// TIA Portal V20 export
TYPE "LKinCtrl_typeSetFlagElement_Bool"
   STRUCT
      flag : Int := -1;   // flag to be set
      flagMode : USInt := 1;   // (see LKinCtrl_PLC_Tags) 0: deactivated; 1: SET_BEFORE_AND_NO_RESET; 2: SET_BEFORE_AND_RESET_AFTER; 3: SET_BEFORE_AND_RESET_AFTER_ONE_CYCLE; 5: SET_BEFORE_AND_NO_RESET_AND_WAIT_FOR_ACKNOWLEDGE; 10: LKINCTRL_FM_SET_AT_REMAINING_DISTANCE; 11: LKINCTRL_FM_SET_AFTER_AND_NO_RESET; 13: LKINCTRL_FM_SET_AFTER_AND_RESET_AFTER_ONE_CYCLE; 15: LKINCTRL_FM_SET_AFTER_AND_NO_RESET_AND_WAIT_FOR_ACKNOWLEDGE
      remainingDistance : LReal := -1.0;   // >0.0: remainingDistance
   END_STRUCT;
END_TYPE
